INTERFACE I_Boiler EXTENDS I_PackML_BaseModule

METHOD Disable : BOOL
VAR_INPUT
END_VAR
END_METHOD

METHOD Enable : BOOL
VAR_INPUT
END_VAR
END_METHOD

PROPERTY Heating : BOOL
GET
END_GET
END_PROPERTY

PROPERTY SetpointMet : BOOL
GET
END_GET
END_PROPERTY

PROPERTY TemperatureSetpoint : LREAL
GET
END_GET
SET
END_SET
END_PROPERTY

END_INTERFACE

(* stored: Version 1.1.0.1
   Itf I_Boiler: Id {7bb3dcbf-7e58-4bf7-852e-ce99eb60453d}
   Method Disable: Id {e58ee186-b71b-46a8-9c8d-ce2eed3e4821}
   Method Enable: Id {729781f5-7167-4206-8c93-370930ef25f7}
   Property Heating: Id {900b263f-bcf5-47e6-b12a-38a87e275572}
   Get Get: Id {b2ae9663-e722-4a55-a432-8d411f44370b}
   Property SetpointMet: Id {0419e36f-9dbe-4be9-9c07-37d931d526dc}
   Get Get: Id {127359cf-0f02-47cf-9e7d-12d731e5a93f}
   Property TemperatureSetpoint: Id {03ce042e-5e11-425c-9a9e-49213f5c14ff}
   Get Get: Id {6e1dcc65-891d-45ef-a042-548d9db4cf0e}
   Set Set: Id {8ec04ad5-ddc1-47bd-beb3-7dc72b1e4125} *)
